FUNCTION_BLOCK Ex70x7_DMC_Channel
VAR_INPUT
END_VAR
VAR_OUTPUT
END_VAR
VAR
	ENCStatus AT%I* : StepperENCStatus;
	STMStatus AT%I* : StepperSTMStatus;
	POSStatus AT%I* : StepperPOSStatus;
	
	ENCControl AT%Q* : StepperENCControl;
	STMControl AT%Q* : StepperSTMControl;
	POSControl AT%Q* : StepperPOSControl;
	
	_InTarget : BOOL;
	
	State :(
		_00_mWait,
        _01_mReset,
        _02_mEnable,
		_06_mGotoPosition,
		_07_mStop,
		_08_mSetPosition,
		_09_RunAtExternalVelo,
		_10_Disable);
		
	tonHoldHigh				: ton;
END_VAR

CASE State OF
        _00_mWait : 
			;
        _01_mReset : 
			STMControl.Reset := TRUE;
			tonHoldHigh(in := TRUE, pt := T#500MS);
			IF tonHoldHigh.Q THEN
				STMControl.Reset := FALSE;
				IF STMStatus.Error = FALSE AND
					STMStatus.Warning = FALSE AND
					STMStatus.Ready = TRUE
				THEN
					State := _00_mWait;
					tonHoldHigh(in := FALSE, pt := T#500MS);
				END_IF
			END_IF
			
        _02_mEnable : 
			IF STMStatus.Error THEN				
				State := _01_mReset;
			ELSE
				STMControl.Enable := TRUE;			
			END_IF
			
		_06_mGotoPosition :
			POSControl.Execute := TRUE;
			_InTarget := FALSE;
			IF POSStatus.InTarget THEN
				State := _02_mEnable;
				POSControl.Execute := FALSE;
				_InTarget := TRUE;
			END_IF
			
		_07_mStop : 
			POSControl.Execute := FALSE;
			IF POSStatus.ReadyToExecute THEN	
				State := _02_mEnable;
			END_IF
			
		_08_mSetPosition :
			POSControl.Execute := TRUE;
			
			IF POSStatus.Calibrated THEN
				POSControl.Execute := FALSE;
				State := _02_mEnable;
			END_IF
			
		_09_RunAtExternalVelo :
			POSControl.Execute := TRUE;
			_InTarget := false;
			
		_10_Disable:
			STMControl.Enable := FALSE;
			State := _00_mWait;
		
			
END_CASE

PROPERTY ActualPosition : lreal
GET
ActualPosition := UDINT_TO_LREAL( POSStatus.ActualPosition)/8062.72;
END_GET
END_PROPERTY

PROPERTY ActualVelocity : int
GET
ActualVelocity := POSStatus.ActualVelocity;
END_GET
END_PROPERTY

METHOD CalibrateMotor : BOOL
VAR_INPUT
END_VAR
IF State = _02_mEnable THEN
	State := _08_mSetPosition;
	//POSControl.Velocity := REAL_TO_INT( Velocity*252);
	POSControl.StartType := StartType.Calibrate;
	//POSControl.TargetPosition := LREAL_TO_UDINT(Position*8062.72);
	//POSControl.TargetPosition := LREAL_TO_UDINT(Position*10);
END_IF
END_METHOD

METHOD Disable : BOOL
VAR_INPUT
END_VAR
IF STMStatus.Ready THEN
	State := _10_Disable;
END_IF
END_METHOD

METHOD Enable : BOOL
VAR_INPUT
END_VAR
IF STMStatus.ReadyToEnable THEN
	State := _02_mEnable;
END_IF
END_METHOD

METHOD GoToPosition : BOOL
VAR_INPUT
	Position : LREAL;
	Velocity : REAL;
END_VAR
IF State = _02_mEnable THEN
	State := _06_mGoToPosition;
	POSControl.Velocity := REAL_TO_INT( Velocity*252);
	POSControl.StartType := StartType.Absolute;
	POSControl.TargetPosition := LREAL_TO_UDINT(Position*8062.72);
END_IF
END_METHOD

PROPERTY InTarget : bool
GET
InTarget := _InTarget;
END_GET
END_PROPERTY

METHOD MoveAtVelocity : BOOL
VAR_INPUT
	Velocity : REAL;
END_VAR
IF State = _02_mEnable THEN
	State := _09_RunAtExternalVelo;
	POSControl.Velocity := REAL_TO_INT( Velocity*252);
	POSControl.StartType := StartType.VeloPositive;
END_IF
END_METHOD

PROPERTY Ready : bool
GET
Ready := STMStatus.Ready;
END_GET
END_PROPERTY

METHOD Reset : BOOL
VAR_INPUT
END_VAR
IF STMStatus.Error OR STMStatus.Warning OR POSStatus.Error THEN
	State := _01_mReset;
END_IF
END_METHOD

METHOD Stop : BOOL
VAR_INPUT
END_VAR
IF POSControl.Execute THEN
	State  := _07_mStop;
END_IF
END_METHOD

END_FUNCTION_BLOCK

(* stored: Version 1.1.0.1, ProductVersion 3.1.4024.9
   POU Ex70x7_DMC_Channel: Id {8dba2e1e-efa3-425a-8683-d8d3e6e0c375}, SpecialFunc None
   Property ActualPosition: Id {e3fd5802-8896-4525-8631-f5b3196112be}
   Get Get: Id {45da7488-4b5c-4824-83e6-ad8e7a921449}
   Property ActualVelocity: Id {39f8e4a8-2a6e-44b9-a7fb-5cc3247407b4}
   Get Get: Id {806c6fd8-5fc9-4c17-9bee-237bb2443294}
   Method CalibrateMotor: Id {869d3233-f21b-441a-9699-57c4eebac93e}
   Method Disable: Id {1be03c52-faf0-4da1-a0b2-99dc1a59ccd4}
   Method Enable: Id {7e2d5fb7-ad9e-4739-a736-c7dd9855344c}
   Method GoToPosition: Id {0a3d70c7-ae77-4ef7-8b45-807a35d4fe22}
   Property InTarget: Id {1a0bd8d2-1200-4f18-9394-803a8831fce4}
   Get Get: Id {a2eca4b5-b96c-4ff4-b68a-669cb9837a01}
   Method MoveAtVelocity: Id {b6daaa03-5be8-4a6b-b2d4-103b287da30a}
   Property Ready: Id {bb0cd970-a59e-4064-a89b-f79082fe5f77}
   Get Get: Id {92b6bcad-3049-41c5-b54d-52bb02cb7445}
   Method Reset: Id {bc8ab3f0-f3f7-4857-b8b2-6bb111ef1733}
   Method Stop: Id {a2ec7f6f-8707-48d8-8908-bb705b2f2285} *)
